TYPE "MEStoPLC_ST350"
VERSION : 0.1
   STRUCT
      Common : "MEStoPLC_Common";
      MainCheckIn : "MEStoPLC_MainCheckIn";
      SubCheckIn : "MEStoPLC_SubCheckIn";
      Processing : "MEStoPLC_ProcessingExchange";
      MainCheckOut : "MEStoPLC_MainCheckOut";
      PrintExchange : "MEStoPLC_PrintExchange";
      AGVExchange : "MEStoPLC_AGVExchange";
      RecipeData : "MEStoPLC_RecipeData_OP220";
   END_STRUCT;

END_TYPE

